TYPE TFMachineTransportManCmd :
STRUCT
END_STRUCT
END_TYPE

(* stored: Version 1.1.0.1, ProductVersion 3.1.4024.11
   DUT TFMachineTransportManCmd: Id {3c95c776-d6f9-4451-80e3-6a031653cb0e} *)
